VAR_GLOBAL
END_VAR
VAR_GLOBAL CONSTANT
	NumOfEcMasters			:UDINT:=6;
END_VAR

(* stored: Version 1.1.0.1, ProductVersion 3.1.4024.11
   GVL GVL: Id {adbe5732-a9a2-4cc5-b700-69ee279e4e4e} *)
